FUNCTION_BLOCK FB_CheckJack2_2
(*
	Description 	: Bloc fonction de test d'un vérin 1 commande, 2 capteurs
	Auteur		: DLA
	Date		: 26.03.2014
	Version		: 1.00

	Modifications :

*)
VAR_INPUT
	bJackGoIn	: BOOL;
	bJackGoOut	: BOOL;
	bJackIsIn	: BOOL;
	bJackIsOut	: BOOL;
	bResetErrors 	: BOOL;
	tTimeOut		: TIME			:= T#400ms;
END_VAR
VAR_OUTPUT
	bJackError	: BOOL;
END_VAR
VAR
	T_Error		: TON;
	RSJackErr	: RS;
	bJackErr		: BOOL;
END_VAR

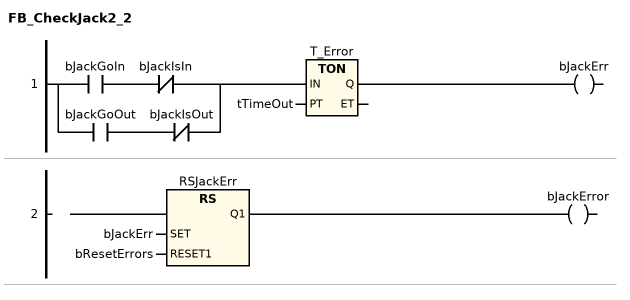
// NETWORK 1
T_Error(IN := bJackGoIn AND NOT bJackIsIn OR bJackGoOut AND NOT bJackIsOut, PT := tTimeOut); // TON
bJackErr := T_Error.Q;

// NETWORK 2
RSJackErr(SET := bJackErr, RESET1 := bResetErrors); // RS
bJackError := RSJackErr.Q1;

END_FUNCTION_BLOCK

(* stored: Version 1.1.0.1, ProductVersion 3.1.4022.12
   POU FB_CheckJack2_2: Id {288a0b36-ddd7-44b5-a074-bb9ea392e392}, SpecialFunc None *)
